(* IEC 61131-3 sources: std_i2980_v2.06_cp053/Source/IMM/ieccontrol/AutoPurgeGeneral, 3 files *)

(* ---- ABManualButton.pu ---- *)
(*

This postupdate algorithm reacts on changes of the autopurge button.
*)

IMPORT_OVER_LISTFILE
 cCompInjection
, tsMoveData
, FBManualButtonKeep
, tevPanelButtonRegister
, tsDeviceId
, tyPanelButton
, tevPanelButtonRegisterData
, tsPanelButton
, FBCheckReady

END_IMPORT

ALGORITHM_BLOCK ABManualButton #DUMMY_EDIT_BLOCK

SYSTEM_VAR
 sv_MoveAutoPurge : tsMoveData;
 di_ButtonAutoPurge : BOOL;
 sv_bInitStart : BOOL;
 sv_bButtonAutoPurge : BOOL;
 sv_bDeviceReady : BOOL;
 sv_bHMILedAutoPurge_ledAttr : BYTE (* Panel LED Attr *);
 sv_bHMILedAutoPurge : BOOL;
 sv_bLedAutoPurge_ledAttr : BYTE (* Panel LED Attr *);
 sv_bLedAutoPurge : BOOL;
 sv_bInitDone : BOOL;
 di_ButtonGeneral1 : BOOL;
 di_ButtonGeneral2 : BOOL;
 sv_iPanelMovementSelector : DINT;
 sv_DeviceId : tsDeviceId;
 sv_PanelButtons : tyPanelButton;
END_VAR

SYSTEM_OBJECT
 PU_Task_7 : TASK;
 PU_Task_13 : TASK;
 evPanelButtonRegister : tevPanelButtonRegister;
END_OBJECT

VAR
 fbManualButton : FBManualButtonKeep;
 mpbInjectionUnitReady : REFTO BOOL;
 evPanelButtonRegisterData : tevPanelButtonRegisterData;
 mpbButtonGeneralAutoPurge1 : REFTO BOOL;
 mpbButtonGeneralAutoPurge2 : REFTO BOOL;
 mbDIButtonAutoPurgeLinked : BOOL;
 mbDIButtonGeneral1Linked : BOOL;
 mbDIButtonGeneral2Linked : BOOL;
 mpiPanelMovementSelector : REFTO DINT;
END_VAR

VAR CONSTANT
 cButtonAutoPurge : DINT := 1;
END_VAR

ALGORITHM aButtonAutoPurge

VAR_INPUT
 bButton : BOOL;
END_VAR
#BEGIN_EDIT_BLOCK
(**************************************** WARNING ********************************************
 *** The KEBA Kemro K2 System including software is not intended for safety control tasks! ***
 ***                       For further information see Comment tab!                        ***
 *********************************************************************************************)

IF bButton AND sv_bDeviceReady AND mpbInjectionUnitReady <> EMPTY AND NOT mpbInjectionUnitReady^ THEN
    // purge should be started and movement of injection function unit active -> ignore manual button
    RETURN;
END_IF;

fbManualButton(bButton := bButton, MoveId := sv_MoveAutoPurge.MoveId, MoveDir := sv_MoveAutoPurge.MoveDir);

;#END_EDIT_BLOCK END_ALGORITHM

POSTUPDATE_ALGORITHM pButtonAutoPurge ON PU_Task_7 WITH di_ButtonAutoPurge,sv_bButtonAutoPurge,mpbButtonGeneralAutoPurge1^,mpbButtonGeneralAutoPurge2^

VAR
 bButton : BOOL;
END_VAR
#BEGIN_EDIT_BLOCK
(**************************************** WARNING ********************************************
 *** The KEBA Kemro K2 System including software is not intended for safety control tasks! ***
 ***                       For further information see Comment tab!                        ***
 *********************************************************************************************)

// soft panel button
bButton := sv_bButtonAutoPurge;

// hw panel button
IF mbDIButtonAutoPurgeLinked THEN
    bButton := bButton OR di_ButtonAutoPurge;
END_IF;

// external panel button
IF CHECK_REF(mpbButtonGeneralAutoPurge1^) THEN
    bButton := bButton OR mpbButtonGeneralAutoPurge1^;
END_IF;
IF CHECK_REF(mpbButtonGeneralAutoPurge2^) THEN
    bButton := bButton OR mpbButtonGeneralAutoPurge2^;
END_IF;

aButtonAutoPurge(bButton := bButton);

;#END_EDIT_BLOCK END_ALGORITHM

POSTUPDATE_ALGORITHM pRegisterButtons ON PU_Task_13 WITH sv_bInitStart

#BEGIN_EDIT_BLOCK
(**************************************** WARNING ********************************************
 *** The KEBA Kemro K2 System including software is not intended for safety control tasks! ***
 ***                       For further information see Comment tab!                        ***
 *********************************************************************************************)

mpbButtonGeneralAutoPurge1 := EMPTY;
mpbButtonGeneralAutoPurge2 := EMPTY;

mbDIButtonAutoPurgeLinked := IS_LINKED(di_ButtonAutoPurge);

mbDIButtonGeneral1Linked := IS_LINKED(di_ButtonGeneral1);
mbDIButtonGeneral2Linked := IS_LINKED(di_ButtonGeneral2);
IF (mbDIButtonGeneral1Linked AND mbDIButtonGeneral2Linked) THEN
    mpiPanelMovementSelector := @sv_iPanelMovementSelector;
END_IF;

evPanelButtonRegisterData.Button.nPanelButtonType := nPanelButtonMovement;
evPanelButtonRegisterData.Button.iCompId := sv_DeviceId.CompId;
evPanelButtonRegisterData.Button.iIndexId := sv_DeviceId.IndexId;
evPanelButtonRegisterData.Button.iButtonId := cButtonAutoPurge;
evPanelButtonRegisterData.Button.pbActionVar1 := @sv_bButtonAutoPurge;
evPanelButtonRegisterData.Button.pbActionVar2 := @sv_bButtonAutoPurge;
evPanelButtonRegisterData.Button.Optional.pbLedVar := @sv_bHMILedAutoPurge;
evPanelButtonRegisterData.Button.Optional.piLedVarAttr := @sv_bHMILedAutoPurge_ledAttr;

SET_EVENT(evPanelButtonRegister, evPanelButtonRegisterData);

;#END_EDIT_BLOCK END_ALGORITHM

POSTUPDATE_ALGORITHM pMoveSelectorChanged ON PU_Task_7 WITH mpiPanelMovementSelector^

VAR
 Button : tsPanelButton;
END_VAR
#BEGIN_EDIT_BLOCK
(**************************************** WARNING ********************************************
 *** The KEBA Kemro K2 System including software is not intended for safety control tasks! ***
 ***                       For further information see Comment tab!                        ***
 *********************************************************************************************)

mpbButtonGeneralAutoPurge1 := EMPTY;
mpbButtonGeneralAutoPurge2 := EMPTY;

IF (NOT sv_bDeviceReady) THEN
    // stop active movements
    aButtonAutoPurge(bButton := FALSE);
END_IF;

IF (sv_iPanelMovementSelector > 0) THEN
    Button := sv_PanelButtons[sv_iPanelMovementSelector];
    IF Button.iCompId = sv_DeviceId.CompId AND
        Button.iIndexId = sv_DeviceId.IndexId THEN

        IF Button.iButtonId = cButtonAutoPurge THEN
            mpbButtonGeneralAutoPurge1 := @di_ButtonGeneral1;
            mpbButtonGeneralAutoPurge2 := @di_ButtonGeneral2;
        END_IF;
    END_IF;
END_IF;

;#END_EDIT_BLOCK END_ALGORITHM

POSTUPDATE_ALGORITHM pLedControl ON PU_Task_7 WITH sv_bDeviceReady

VAR
 bInitDone : BOOL;
 mbLedAutoPurgeExists : BOOL := FALSE;
END_VAR
#BEGIN_EDIT_BLOCK
IF NOT bInitDone THEN
    sv_bHMILedAutoPurge_ledAttr := 16#3;
    IF IS_LINKED(sv_bLedAutoPurge) AND IS_LINKED(sv_bLedAutoPurge_ledAttr) THEN
        sv_bLedAutoPurge_ledAttr := sv_bHMILedAutoPurge_ledAttr;
        mbLedAutoPurgeExists := TRUE;
    ELSE
        mbLedAutoPurgeExists := FALSE;
    END_IF;

    bInitDone := TRUE;
END_IF;

IF NOT sv_bDeviceReady THEN
   //led should be on if purging is active
   sv_bHMILedAutoPurge := TRUE;
ELSE
   //switch off
   sv_bHMILedAutoPurge := FALSE;
END_IF;

IF mbLedAutoPurgeExists THEN
   sv_bLedAutoPurge := sv_bHMILedAutoPurge;
END_IF;

;#END_EDIT_BLOCK END_ALGORITHM

POSTUPDATE_ALGORITHM pInitDone ON PU_Task_7(10) WITH sv_bInitDone

VAR
 fbCheckInjectionReady : FBCheckReady;
 DeviceIdInjection : tsDeviceId;
END_VAR
#BEGIN_EDIT_BLOCK
(**************************************** WARNING ********************************************
 *** The KEBA Kemro K2 System including software is not intended for safety control tasks! ***
 ***                       For further information see Comment tab!                        ***
 *********************************************************************************************)

//get reference to ready flag of injection function unit
DeviceIdInjection.CompId := cCompInjection;
DeviceIdInjection.IndexId := sv_DeviceId.IndexId;

fbCheckInjectionReady(DeviceId := DeviceIdInjection);
mpbInjectionUnitReady := fbCheckInjectionReady.pbReady;

;#END_EDIT_BLOCK END_ALGORITHM

END_ALGORITHM_BLOCK

#END_OF_IEC_PART

@Puma @IecEditor 6 114 @Pou 25
@@@BEG_Comment@@@

This postupdate algorithm reacts on changes of the autopurge button.
@@@END_Comment@@@

@BEG_Contents

@BEG_Func
@RT(17)FuncTreeContainer
0
@END_Func

@BEG_Const
@RT(18)ConstTreeContainer
1
@Var @RT(14)cCompInjection @RT(0) @T @F @DT @RT(4)DINT @RT(0) @T @T @BASIC 0 @F
@F @F
@T
@BEG_Attrib
0 @RT(3)104 @RT(19)Component Injection
@END_Attrib
1 1 @F @F @F @F

@END_Const

@BEG_Export

@BEG_Kind
@ALGORITHM_BLOCK @RT(14)ABManualButton @STRUCTURED_TEXT
@RT(0) @RT(0) @RT(0)
@END_Kind

@BEG_Dcl
@RT(16)DclTreeContainer
28
@Var @RT(16)sv_MoveAutoPurge @RT(0) @T @T @DERIVED 0 @T @T @DT @RT(10)tsMoveData @RT(0) @T @T @UNKNOWN 0 @F
@F @F
@T
@BEG_Attrib
3 @RT(0) @RT(0) @RT(0)
@END_Attrib
1 8 @F @F @F @F

@Var @RT(18)di_ButtonAutoPurge @RT(0) @T @F @DT @RT(4)BOOL @RT(0) @T @T @BASIC 0 @F
@F @F
@T
@BEG_Attrib
3 @RT(0) @RT(0) @RT(0)
@END_Attrib
1 8 @F @F @F @F

@Var @RT(13)sv_bInitStart @RT(0) @T @F @DT @RT(4)BOOL @RT(0) @T @T @BASIC 0 @F
@F @F
@T
@BEG_Attrib
3 @RT(0) @RT(0) @RT(0)
@END_Attrib
1 8 @F @F @F @F

@Var @RT(19)sv_bButtonAutoPurge @RT(0) @T @F @DT @RT(4)BOOL @RT(0) @T @T @BASIC 0 @F
@F @F
@T
@BEG_Attrib
3 @RT(0) @RT(0) @RT(0)
@END_Attrib
1 8 @F @F @F @F

@Var @RT(15)sv_bDeviceReady @RT(0) @T @F @DT @RT(4)BOOL @RT(0) @T @T @BASIC 0 @F
@F @F
@T
@BEG_Attrib
3 @RT(0) @RT(0) @RT(0)
@END_Attrib
1 8 @F @F @F @F

@Var @RT(27)sv_bHMILedAutoPurge_ledAttr @RT(0) @T @F @DT @RT(4)BYTE @RT(0) @T @T @BASIC 0 @F
@F @F
@T
@BEG_Attrib
3 @RT(0) @RT(14)Panel LED Attr @RT(0)
@END_Attrib
1 8 @F @F @F @F

@Var @RT(19)sv_bHMILedAutoPurge @RT(0) @T @F @DT @RT(4)BOOL @RT(0) @T @T @BASIC 0 @F
@F @F
@T
@BEG_Attrib
3 @RT(0) @RT(0) @RT(0)
@END_Attrib
1 8 @F @F @F @F

@Var @RT(24)sv_bLedAutoPurge_ledAttr @RT(0) @T @F @DT @RT(4)BYTE @RT(0) @T @T @BASIC 0 @F
@F @F
@T
@BEG_Attrib
3 @RT(0) @RT(14)Panel LED Attr @RT(0)
@END_Attrib
1 8 @F @F @F @F

@Var @RT(16)sv_bLedAutoPurge @RT(0) @T @F @DT @RT(4)BOOL @RT(0) @T @T @BASIC 0 @F
@F @F
@T
@BEG_Attrib
3 @RT(0) @RT(0) @RT(0)
@END_Attrib
1 8 @F @F @F @F

@Var @RT(12)sv_bInitDone @RT(0) @T @F @DT @RT(4)BOOL @RT(0) @T @T @BASIC 0 @F
@F @F
@T
@BEG_Attrib
3 @RT(0) @RT(0) @RT(0)
@END_Attrib
1 8 @F @F @F @F

@Var @RT(9)PU_Task_7 @RT(0) @T @F @DT @RT(4)TASK @RT(0) @T @T @BASIC 0 @F
@F @F
@T
@BEG_Attrib
3 @RT(0) @RT(0) @RT(0)
@END_Attrib
1 7 @F @F @F @F

@Var @RT(10)PU_Task_13 @RT(0) @T @F @DT @RT(4)TASK @RT(0) @T @T @BASIC 0 @F
@F @F
@T
@BEG_Attrib
3 @RT(0) @RT(0) @RT(0)
@END_Attrib
1 7 @F @F @F @F

@Var @RT(14)fbManualButton @RT(0) @T @T @DERIVED 0 @T @T @DT @RT(18)FBManualButtonKeep @RT(0) @T @T @UNKNOWN 0 @F
@F @F
@T
@BEG_Attrib
3 @RT(0) @RT(0) @RT(0)
@END_Attrib
1 0 @F @F @F @F

@Var @RT(21)mpbInjectionUnitReady @RT(0) @T @T @REFTO 0 @T @DT @RT(4)BOOL @RT(0) @T @T @BASIC 0 @F
@F @F
@T
@BEG_Attrib
3 @RT(0) @RT(0) @RT(0)
@END_Attrib
1 0 @F @F @F @F

@Var @RT(21)evPanelButtonRegister @RT(0) @T @T @DERIVED 0 @T @T @DT @RT(22)tevPanelButtonRegister @RT(0) @T @T @UNKNOWN 0 @F
@F @F
@T
@BEG_Attrib
3 @RT(0) @RT(0) @RT(0)
@END_Attrib
1 7 @F @F @F @F

@Var @RT(17)di_ButtonGeneral1 @RT(0) @T @F @DT @RT(4)BOOL @RT(0) @T @T @BASIC 0 @F
@F @F
@T
@BEG_Attrib
3 @RT(0) @RT(0) @RT(0)
@END_Attrib
1 8 @F @F @F @F

@Var @RT(17)di_ButtonGeneral2 @RT(0) @T @F @DT @RT(4)BOOL @RT(0) @T @T @BASIC 0 @F
@F @F
@T
@BEG_Attrib
3 @RT(0) @RT(0) @RT(0)
@END_Attrib
1 8 @F @F @F @F

@Var @RT(25)sv_iPanelMovementSelector @RT(0) @T @F @DT @RT(4)DINT @RT(0) @T @T @BASIC 0 @F
@F @F
@T
@BEG_Attrib
3 @RT(0) @RT(0) @RT(0)
@END_Attrib
1 8 @F @F @F @F

@Var @RT(11)sv_DeviceId @RT(0) @T @T @DERIVED 0 @T @T @DT @RT(10)tsDeviceId @RT(0) @T @T @UNKNOWN 0 @F
@F @F
@T
@BEG_Attrib
3 @RT(0) @RT(0) @RT(0)
@END_Attrib
1 8 @F @F @F @F

@Var @RT(15)sv_PanelButtons @RT(0) @T @T @DERIVED 0 @T @T @DT @RT(13)tyPanelButton @RT(0) @T @T @UNKNOWN 0 @F
@F @F
@T
@BEG_Attrib
3 @RT(0) @RT(0) @RT(0)
@END_Attrib
1 8 @F @F @F @F

@Var @RT(25)evPanelButtonRegisterData @RT(0) @T @T @DERIVED 0 @T @T @DT @RT(26)tevPanelButtonRegisterData @RT(0) @T @T @UNKNOWN 0 @F
@F @F
@T
@BEG_Attrib
3 @RT(0) @RT(0) @RT(0)
@END_Attrib
1 0 @F @F @F @F

@Var @RT(26)mpbButtonGeneralAutoPurge1 @RT(0) @T @T @REFTO 0 @T @DT @RT(4)BOOL @RT(0) @T @T @BASIC 0 @F
@F @F
@T
@BEG_Attrib
3 @RT(0) @RT(0) @RT(0)
@END_Attrib
1 0 @F @F @F @F

@Var @RT(26)mpbButtonGeneralAutoPurge2 @RT(0) @T @T @REFTO 0 @T @DT @RT(4)BOOL @RT(0) @T @T @BASIC 0 @F
@F @F
@T
@BEG_Attrib
3 @RT(0) @RT(0) @RT(0)
@END_Attrib
1 0 @F @F @F @F

@Var @RT(25)mbDIButtonAutoPurgeLinked @RT(0) @T @F @DT @RT(4)BOOL @RT(0) @T @T @BASIC 0 @F
@F @F
@T
@BEG_Attrib
3 @RT(0) @RT(0) @RT(0)
@END_Attrib
1 0 @F @F @F @F

@Var @RT(24)mbDIButtonGeneral1Linked @RT(0) @T @F @DT @RT(4)BOOL @RT(0) @T @T @BASIC 0 @F
@F @F
@T
@BEG_Attrib
3 @RT(0) @RT(0) @RT(0)
@END_Attrib
1 0 @F @F @F @F

@Var @RT(24)mbDIButtonGeneral2Linked @RT(0) @T @F @DT @RT(4)BOOL @RT(0) @T @T @BASIC 0 @F
@F @F
@T
@BEG_Attrib
3 @RT(0) @RT(0) @RT(0)
@END_Attrib
1 0 @F @F @F @F

@Var @RT(16)cButtonAutoPurge @RT(0) @T @F @DT @RT(4)DINT @RT(0) @T @T @BASIC 0 @F
@F @F
@T
@BEG_Attrib
3 @RT(1)1 @RT(0) @RT(0)
@END_Attrib
1 15 @F @F @F @F

@Var @RT(24)mpiPanelMovementSelector @RT(0) @T @T @REFTO 0 @T @DT @RT(4)DINT @RT(0) @T @T @BASIC 0 @F
@F @F
@T
@BEG_Attrib
3 @RT(0) @RT(0) @RT(0)
@END_Attrib
1 0 @F @F @F @F

@END_Dcl

@END_Export

@BEG_Body

6

@BEG_Export

@BEG_Algo
@ALGORITHM @RT(16)aButtonAutoPurge @STRUCTURED_TEXT
@RT(0) @RT(0) @RT(0) @F @F
@END_Algo

@BEG_Dcl
@RT(16)DclTreeContainer
1
@Var @RT(7)bButton @RT(0) @T @F @DT @RT(4)BOOL @RT(0) @T @T @BASIC 0 @F
@F @F
@T
@BEG_Attrib
3 @RT(0) @RT(0) @RT(0)
@END_Attrib
1 1 @F @F @F @F

@END_Dcl

@END_Export

@BEG_Export

@BEG_Algo
@POSTUPDATE_ALGORITHM @RT(16)pButtonAutoPurge @STRUCTURED_TEXT
@RT(0) @RT(94)di_ButtonAutoPurge,sv_bButtonAutoPurge,mpbButtonGeneralAutoPurge1^,mpbButtonGeneralAutoPurge2^ @RT(9)PU_Task_7 @F @F
@END_Algo

@BEG_Dcl
@RT(16)DclTreeContainer
1
@Var @RT(7)bButton @RT(0) @T @F @DT @RT(4)BOOL @RT(0) @T @T @BASIC 0 @F
@F @F
@T
@BEG_Attrib
3 @RT(0) @RT(0) @RT(0)
@END_Attrib
1 0 @F @F @F @F

@END_Dcl

@END_Export

@BEG_Export

@BEG_Algo
@POSTUPDATE_ALGORITHM @RT(16)pRegisterButtons @STRUCTURED_TEXT
@RT(0) @RT(13)sv_bInitStart @RT(10)PU_Task_13 @F @F
@END_Algo

@BEG_Dcl
@RT(16)DclTreeContainer
0
@END_Dcl

@END_Export

@BEG_Export

@BEG_Algo
@POSTUPDATE_ALGORITHM @RT(20)pMoveSelectorChanged @STRUCTURED_TEXT
@RT(0) @RT(25)mpiPanelMovementSelector^ @RT(9)PU_Task_7 @F @F
@END_Algo

@BEG_Dcl
@RT(16)DclTreeContainer
1
@Var @RT(6)Button @RT(0) @T @T @DERIVED 0 @T @T @DT @RT(13)tsPanelButton @RT(0) @T @T @UNKNOWN 0 @F
@F @F
@T
@BEG_Attrib
3 @RT(0) @RT(0) @RT(0)
@END_Attrib
1 0 @F @F @F @F

@END_Dcl

@END_Export

@BEG_Export

@BEG_Algo
@POSTUPDATE_ALGORITHM @RT(11)pLedControl @STRUCTURED_TEXT
@RT(0) @RT(15)sv_bDeviceReady @RT(9)PU_Task_7 @F @F
@END_Algo

@BEG_Dcl
@RT(16)DclTreeContainer
2
@Var @RT(9)bInitDone @RT(0) @T @F @DT @RT(4)BOOL @RT(0) @T @T @BASIC 0 @F
@F @F
@T
@BEG_Attrib
3 @RT(0) @RT(0) @RT(0)
@END_Attrib
1 0 @F @F @F @F

@Var @RT(20)mbLedAutoPurgeExists @RT(0) @T @F @DT @RT(4)BOOL @RT(0) @T @T @BASIC 0 @F
@F @F
@T
@BEG_Attrib
3 @RT(5)FALSE @RT(0) @RT(0)
@END_Attrib
1 0 @F @F @F @F

@END_Dcl

@END_Export

@BEG_Export

@BEG_Algo
@POSTUPDATE_ALGORITHM @RT(9)pInitDone @STRUCTURED_TEXT
@RT(0) @RT(12)sv_bInitDone @RT(13)PU_Task_7(10) @F @F
@END_Algo

@BEG_Dcl
@RT(16)DclTreeContainer
2
@Var @RT(21)fbCheckInjectionReady @RT(0) @T @T @DERIVED 0 @T @T @DT @RT(12)FBCheckReady @RT(0) @T @T @UNKNOWN 0 @F
@F @F
@T
@BEG_Attrib
3 @RT(0) @RT(0) @RT(0)
@END_Attrib
1 0 @F @F @F @F

@Var @RT(17)DeviceIdInjection @RT(0) @T @T @DERIVED 0 @T @T @DT @RT(10)tsDeviceId @RT(0) @T @T @UNKNOWN 0 @F
@F @F
@T
@BEG_Attrib
3 @RT(0) @RT(0) @RT(0)
@END_Attrib
1 0 @F @F @F @F

@END_Dcl

@END_Export

@BEG_Body
@TL(13)
(**************************************** WARNING ********************************************
 *** The KEBA Kemro K2 System including software is not intended for safety control tasks! ***
 ***                       For further information see Comment tab!                        ***
 *********************************************************************************************)

IF bButton AND sv_bDeviceReady AND mpbInjectionUnitReady <> EMPTY AND NOT mpbInjectionUnitReady^ THEN
    // purge should be started and movement of injection function unit active -> ignore manual button
    RETURN;
END_IF;

fbManualButton(bButton := bButton, MoveId := sv_MoveAutoPurge.MoveId, MoveDir := sv_MoveAutoPurge.MoveDir);

@END_Body

@@@BEG_Comment@@@
@TL(0)

@@@END_Comment@@@

@BEG_Body
@TL(24)
(**************************************** WARNING ********************************************
 *** The KEBA Kemro K2 System including software is not intended for safety control tasks! ***
 ***                       For further information see Comment tab!                        ***
 *********************************************************************************************)

// soft panel button
bButton := sv_bButtonAutoPurge;

// hw panel button
IF mbDIButtonAutoPurgeLinked THEN
    bButton := bButton OR di_ButtonAutoPurge;
END_IF;

// external panel button
IF CHECK_REF(mpbButtonGeneralAutoPurge1^) THEN
    bButton := bButton OR mpbButtonGeneralAutoPurge1^;
END_IF;
IF CHECK_REF(mpbButtonGeneralAutoPurge2^) THEN
    bButton := bButton OR mpbButtonGeneralAutoPurge2^;
END_IF;

aButtonAutoPurge(bButton := bButton);

@END_Body

@@@BEG_Comment@@@
@TL(0)

@@@END_Comment@@@

@BEG_Body
@TL(27)
(**************************************** WARNING ********************************************
 *** The KEBA Kemro K2 System including software is not intended for safety control tasks! ***
 ***                       For further information see Comment tab!                        ***
 *********************************************************************************************)

mpbButtonGeneralAutoPurge1 := EMPTY;
mpbButtonGeneralAutoPurge2 := EMPTY;

mbDIButtonAutoPurgeLinked := IS_LINKED(di_ButtonAutoPurge);

mbDIButtonGeneral1Linked := IS_LINKED(di_ButtonGeneral1);
mbDIButtonGeneral2Linked := IS_LINKED(di_ButtonGeneral2);
IF (mbDIButtonGeneral1Linked AND mbDIButtonGeneral2Linked) THEN
    mpiPanelMovementSelector := @sv_iPanelMovementSelector;
END_IF;

evPanelButtonRegisterData.Button.nPanelButtonType := nPanelButtonMovement;
evPanelButtonRegisterData.Button.iCompId := sv_DeviceId.CompId;
evPanelButtonRegisterData.Button.iIndexId := sv_DeviceId.IndexId;
evPanelButtonRegisterData.Button.iButtonId := cButtonAutoPurge;
evPanelButtonRegisterData.Button.pbActionVar1 := @sv_bButtonAutoPurge;
evPanelButtonRegisterData.Button.pbActionVar2 := @sv_bButtonAutoPurge;
evPanelButtonRegisterData.Button.Optional.pbLedVar := @sv_bHMILedAutoPurge;
evPanelButtonRegisterData.Button.Optional.piLedVarAttr := @sv_bHMILedAutoPurge_ledAttr;

SET_EVENT(evPanelButtonRegister, evPanelButtonRegisterData);

@END_Body

@@@BEG_Comment@@@
@TL(0)

@@@END_Comment@@@

@BEG_Body
@TL(26)
(**************************************** WARNING ********************************************
 *** The KEBA Kemro K2 System including software is not intended for safety control tasks! ***
 ***                       For further information see Comment tab!                        ***
 *********************************************************************************************)

mpbButtonGeneralAutoPurge1 := EMPTY;
mpbButtonGeneralAutoPurge2 := EMPTY;

IF (NOT sv_bDeviceReady) THEN
    // stop active movements
    aButtonAutoPurge(bButton := FALSE);
END_IF;

IF (sv_iPanelMovementSelector > 0) THEN
    Button := sv_PanelButtons[sv_iPanelMovementSelector];
    IF Button.iCompId = sv_DeviceId.CompId AND
        Button.iIndexId = sv_DeviceId.IndexId THEN

        IF Button.iButtonId = cButtonAutoPurge THEN
            mpbButtonGeneralAutoPurge1 := @di_ButtonGeneral1;
            mpbButtonGeneralAutoPurge2 := @di_ButtonGeneral2;
        END_IF;
    END_IF;
END_IF;

@END_Body

@@@BEG_Comment@@@
@TL(0)

@@@END_Comment@@@

@BEG_Body
@TL(26)
IF NOT bInitDone THEN
    sv_bHMILedAutoPurge_ledAttr := 16#3;
    IF IS_LINKED(sv_bLedAutoPurge) AND IS_LINKED(sv_bLedAutoPurge_ledAttr) THEN
        sv_bLedAutoPurge_ledAttr := sv_bHMILedAutoPurge_ledAttr;
        mbLedAutoPurgeExists := TRUE;
    ELSE
        mbLedAutoPurgeExists := FALSE;
    END_IF;

    bInitDone := TRUE;
END_IF;

IF NOT sv_bDeviceReady THEN
   //led should be on if purging is active
   sv_bHMILedAutoPurge := TRUE;
ELSE
   //switch off
   sv_bHMILedAutoPurge := FALSE;
END_IF;

IF mbLedAutoPurgeExists THEN
   sv_bLedAutoPurge := sv_bHMILedAutoPurge;
END_IF;

@END_Body

@@@BEG_Comment@@@
@TL(0)

@@@END_Comment@@@

@BEG_Body
@TL(13)
(**************************************** WARNING ********************************************
 *** The KEBA Kemro K2 System including software is not intended for safety control tasks! ***
 ***                       For further information see Comment tab!                        ***
 *********************************************************************************************)

//get reference to ready flag of injection function unit
DeviceIdInjection.CompId := cCompInjection;
DeviceIdInjection.IndexId := sv_DeviceId.IndexId;

fbCheckInjectionReady(DeviceId := DeviceIdInjection);
mpbInjectionUnitReady := fbCheckInjectionReady.pbReady;

@END_Body

@@@BEG_Comment@@@
@TL(0)

@@@END_Comment@@@
@END_Body

@END_Contents

(* ---- ABMoveAutoPurge.pu ---- *)
(*

@FunctionID: S_KPIEC_PRINJ_03

*)

IMPORT_OVER_LISTFILE
 SET_EVENT
, cLockGroupHeatingNozzle
, cLockGroupSafetyGateNozzle
, cLockGroupSafetyGateMold
, cLockGroupMotor
, cCompInjection
, cMoveFwd
, cMoveInjectPurge
, cMoveBwd
, cMoveDecompPurge
, cMovePlastPurge
, cCompShutOffNozzle
, cMoveClose
, cMoveOpen
, tsMoveData
, tsPurgeSettings
, tsActPurgeTimes
, tyNumberOfDevices
, tsDeviceId
, tevStartRequest
, ABMovementRegister
, tevStartRequestData
, FBCheckReady
, FBStop
, FBCheckPosReached
, FBDebugTrace2

END_IMPORT

ALGORITHM_BLOCK ABMoveAutoPurge #DUMMY_EDIT_BLOCK

SYSTEM_VAR
 sv_MoveAutoPurge : tsMoveData;
 sv_PurgeSettings : tsPurgeSettings;
 sv_rScrewPosition : REAL (* actual screw position *);
 sv_ActPurgeTimes : tsActPurgeTimes;
 sv_NumberOfDevices : tyNumberOfDevices;
 sv_DeviceId : tsDeviceId;
END_VAR

SYSTEM_OBJECT
 evStartRequest : tevStartRequest;
END_OBJECT

ALGORITHM aRegister

VAR
 abMovementRegister : ABMovementRegister;
END_VAR
#BEGIN_EDIT_BLOCK
(**************************************** WARNING ********************************************
 *** The KEBA Kemro K2 System including software is not intended for safety control tasks! ***
 ***                       For further information see Comment tab!                        ***
 *********************************************************************************************)

// movement registration
sv_MoveAutoPurge.LockGroups[1] := cLockGroupHeatingNozzle;
sv_MoveAutoPurge.LockGroups[2] := cLockGroupSafetyGateNozzle;
sv_MoveAutoPurge.LockGroups[3] := cLockGroupSafetyGateMold;
sv_MoveAutoPurge.LockGroups[4] := cLockGroupMotor;

abMovementRegister.aRegister(@sv_MoveAutoPurge);

;#END_EDIT_BLOCK END_ALGORITHM

ALGORITHM aRun

VAR_OUTPUT
 bReady : BOOL;
END_VAR

VAR_INPUT
 bStop : BOOL;
END_VAR

VAR
 evStartRequestData : tevStartRequestData;
 DeviceId : tsDeviceId;
 fbCheckReady : FBCheckReady;
 iCount : DINT;
 fbStop : FBStop;
 bShutOffNozzleAvailable : BOOL;
 bInitDone : BOOL;
 pbShutOffNozzleOpen : REFTO BOOL;
 pbShutOffNozzleClosed : REFTO BOOL;
 DeviceIdShutOffNozzle : tsDeviceId;
 fbCheckPosReached : FBCheckPosReached;
 fbDebugTrace2 : FBDebugTrace2;
 dTmpPurgePlastTime : TIME;
 rTmpPurgeDecompPos : REAL;
END_VAR

(* IecGraph-Code *)

(* init step *)
INITIAL_STEP S_Start:
AInitShutOffNozzle (P);
AStart (P);
END_STEP

ACTION AStart: #BEGIN_EDIT_BLOCK
bReady := FALSE;
fbDebugTrace2(nDeviceState, 'AutoPurge started');
iCount := 0;

;#END_EDIT_BLOCK END_ACTION (*AStart*)

(* steps *)
STEP Step17:
END_STEP

STEP S_OpenShutOffNozzle:
AStartOpen (P);
ACheckShutOffNozzle (N);
END_STEP

ACTION ACheckShutOffNozzle: #BEGIN_EDIT_BLOCK
fbCheckReady(DeviceId := DeviceId);

;#END_EDIT_BLOCK END_ACTION (*ACheckShutOffNozzle*)
STEP S_Inject:
AStartInject (P);
ACheckInjectReady (N);
END_STEP

ACTION AStartInject: #BEGIN_EDIT_BLOCK
// send start request
DeviceId.CompId := cCompInjection;
DeviceId.IndexId := sv_DeviceId.IndexId;

evStartRequestData.DeviceId := DeviceId;
evStartRequestData.MoveDir := cMoveFwd;
evStartRequestData.MoveId := cMoveInjectPurge;
SET_EVENT(evStartRequest, evStartRequestData);

;#END_EDIT_BLOCK END_ACTION (*AStartInject*)
ACTION ACheckInjectReady: #BEGIN_EDIT_BLOCK
fbCheckReady(DeviceId := DeviceId);

;#END_EDIT_BLOCK END_ACTION (*ACheckInjectReady*)
STEP S_Decomp:
AStartDecomp (P);
ACheckDecompReady (N);
END_STEP

ACTION AStartDecomp: #BEGIN_EDIT_BLOCK
//copy decomp position to avoid wrongly detecting a error
//when the value changes while the movement is active
rTmpPurgeDecompPos := sv_PurgeSettings.DecompParams.rEndPos;

// send start request
DeviceId.CompId := cCompInjection;
DeviceId.IndexId := sv_DeviceId.IndexId;

evStartRequestData.DeviceId := DeviceId;
evStartRequestData.MoveDir := cMoveBwd;
evStartRequestData.MoveId := cMoveDecompPurge;
SET_EVENT(evStartRequest, evStartRequestData);

;#END_EDIT_BLOCK END_ACTION (*AStartDecomp*)
ACTION ACheckDecompReady: #BEGIN_EDIT_BLOCK
fbCheckReady(DeviceId := DeviceId);

;#END_EDIT_BLOCK END_ACTION (*ACheckDecompReady*)
STEP S_Plast:
AStartPlast (P);
ACheckPlastReady (N);
END_STEP

ACTION AStartPlast: #BEGIN_EDIT_BLOCK
//copy purge set time to avoid wrongly detecting a error
//when the value changes while the movement is active
dTmpPurgePlastTime := sv_PurgeSettings.PlastParams.dSetPlastTime;

// send start request
DeviceId.CompId := cCompInjection;
DeviceId.IndexId := sv_DeviceId.IndexId;

evStartRequestData.DeviceId := DeviceId;
evStartRequestData.MoveDir := cMoveBwd;
evStartRequestData.MoveId := cMovePlastPurge;
SET_EVENT(evStartRequest, evStartRequestData);

;#END_EDIT_BLOCK END_ACTION (*AStartPlast*)
ACTION ACheckPlastReady: #BEGIN_EDIT_BLOCK
fbCheckReady(DeviceId := DeviceId);

;#END_EDIT_BLOCK END_ACTION (*ACheckPlastReady*)
STEP S_CheckCounter:
ACounter (P);
END_STEP

ACTION ACounter: #BEGIN_EDIT_BLOCK
iCount := iCount + 1;

;#END_EDIT_BLOCK END_ACTION (*ACounter*)
STEP S_CheckStop:
END_STEP

STEP S_Stop:
AStopActiveMovement (P);
AStoppedMoveReady (N);
END_STEP

ACTION AStopActiveMovement: #BEGIN_EDIT_BLOCK
//stop actual active movement
fbStop(DeviceId := DeviceId);

;#END_EDIT_BLOCK END_ACTION (*AStopActiveMovement*)
ACTION AStoppedMoveReady: #BEGIN_EDIT_BLOCK
fbCheckReady(DeviceId := DeviceId);

;#END_EDIT_BLOCK END_ACTION (*AStoppedMoveReady*)
STEP Step27:
END_STEP

STEP S_CloseShutOffNozzle:
AStartClose (P);
ACheckShutOff (N);
END_STEP

ACTION ACheckShutOff: #BEGIN_EDIT_BLOCK
fbCheckReady(DeviceId := DeviceId);

;#END_EDIT_BLOCK END_ACTION (*ACheckShutOff*)
STEP S_Ready:
AReady (P);
END_STEP

ACTION AReady: #BEGIN_EDIT_BLOCK
bReady := TRUE;
fbDebugTrace2(nDeviceState, 'AutoPurge ready');

;#END_EDIT_BLOCK END_ACTION (*AReady*)

(* transitions *)
GO_ON_TRANSITION TStart (* Trans21 *) FROM S_Start TO Step17 :=  #BEGIN_EDIT_BLOCK
TRUE
;#END_EDIT_BLOCK
END_TRANSITION

GO_ON_TRANSITION TShutOffNozzle (* TShutOffNozzle *) FROM Step17 TO S_OpenShutOffNozzle :=  #BEGIN_EDIT_BLOCK
bShutOffNozzleAvailable
;#END_EDIT_BLOCK
END_TRANSITION

TRANSITION TShutOffNozzleOpen (* TShutOffNozzleOpen *) FROM S_OpenShutOffNozzle TO S_Inject :=  #BEGIN_EDIT_BLOCK
fbCheckReady.bReady AND pbShutOffNozzleOpen^
;#END_EDIT_BLOCK
END_TRANSITION

TRANSITION TStop4 (* TStop4 *) FROM S_OpenShutOffNozzle TO S_Stop :=  #BEGIN_EDIT_BLOCK
bStop
;#END_EDIT_BLOCK
END_TRANSITION

GO_ON_TRANSITION TNoShutOffNozzle (* TNoShutOffNozzle *) FROM Step17 TO S_Inject :=  #BEGIN_EDIT_BLOCK
NOT bShutOffNozzleAvailable
;#END_EDIT_BLOCK
END_TRANSITION

TRANSITION TInjectReady (* TInjectReady *) FROM S_Inject TO S_Decomp :=  #BEGIN_EDIT_BLOCK
fbCheckReady.bReady AND
sv_rScrewPosition <= sv_PurgeSettings.InjectParams.rEndPos
;#END_EDIT_BLOCK
END_TRANSITION

TRANSITION TStop1 (* TStop1 *) FROM S_Inject TO S_Stop :=  #BEGIN_EDIT_BLOCK
bStop
;#END_EDIT_BLOCK
END_TRANSITION

TRANSITION TDecompReady (* TDecompReady *) FROM S_Decomp TO S_Plast :=  #BEGIN_EDIT_BLOCK
fbCheckReady.bReady AND
sv_rScrewPosition >= rTmpPurgeDecompPos
;#END_EDIT_BLOCK
END_TRANSITION

TRANSITION TStop2 (* TStop2 *) FROM S_Decomp TO S_Stop :=  #BEGIN_EDIT_BLOCK
bStop
;#END_EDIT_BLOCK
END_TRANSITION

TRANSITION TPlastReady (* TPlastReady *) FROM S_Plast TO S_CheckCounter :=  #BEGIN_EDIT_BLOCK
fbCheckReady.bReady AND
sv_ActPurgeTimes.dActPlastTime >= dTmpPurgePlastTime
;#END_EDIT_BLOCK
END_TRANSITION

TRANSITION TStop3 (* TStop3 *) FROM S_Plast TO S_Stop :=  #BEGIN_EDIT_BLOCK
bStop
;#END_EDIT_BLOCK
END_TRANSITION

GO_ON_TRANSITION TRepeat (* TRepeat *) FROM S_CheckCounter TO S_Inject :=  #BEGIN_EDIT_BLOCK
iCount < sv_PurgeSettings.iCount
;#END_EDIT_BLOCK
END_TRANSITION

GO_ON_TRANSITION TReady (* TReady *) FROM S_CheckCounter TO S_CheckStop :=  #BEGIN_EDIT_BLOCK
iCount = sv_PurgeSettings.iCount
;#END_EDIT_BLOCK
END_TRANSITION

GO_ON_TRANSITION TStop (* TStop *) FROM S_CheckStop TO S_Stop :=  #BEGIN_EDIT_BLOCK
bStop
;#END_EDIT_BLOCK
END_TRANSITION

TRANSITION TStoppedDeviceReady (* TStoppedDeviceReady *) FROM S_Stop TO Step27 :=  #BEGIN_EDIT_BLOCK
fbCheckReady.bReady
;#END_EDIT_BLOCK
END_TRANSITION

GO_ON_TRANSITION TNoStop (* TNoStop *) FROM S_CheckStop TO Step27 :=  #BEGIN_EDIT_BLOCK
NOT bStop
;#END_EDIT_BLOCK
END_TRANSITION

GO_ON_TRANSITION Trans36 (* Trans36 *) FROM Step27 TO S_CloseShutOffNozzle :=  #BEGIN_EDIT_BLOCK
bShutOffNozzleAvailable
;#END_EDIT_BLOCK
END_TRANSITION

TRANSITION TShutOffNozzleReady (* TShutOffNozzleClosed *) FROM S_CloseShutOffNozzle TO S_Ready :=  #BEGIN_EDIT_BLOCK
fbCheckReady.bReady
;#END_EDIT_BLOCK
END_TRANSITION

GO_ON_TRANSITION Trans37 (* Trans37 *) FROM Step27 TO S_Ready :=  #BEGIN_EDIT_BLOCK
NOT bShutOffNozzleAvailable
;#END_EDIT_BLOCK
END_TRANSITION

TRANSITION Trans12 (* Trans12 *) FROM S_Ready TO S_Start :=  #BEGIN_EDIT_BLOCK
TRUE
;#END_EDIT_BLOCK
END_TRANSITION

(* end IecGraph-Code *)
(* sfc-code *)

(* stand alone actions *)
ACTION AInitShutOffNozzle: #BEGIN_EDIT_BLOCK
//check if shut off nozzle is available
IF NOT bInitDone THEN
   bShutOffNozzleAvailable := sv_NumberOfDevices[cCompShutOffNozzle] = sv_DeviceId.IndexId;
END_IF;

IF bShutOffNozzleAvailable AND NOT bInitDone THEN
   //get pos reached flags of shut off nozzle
   DeviceIdShutOffNozzle.CompId := cCompShutOffNozzle;
   DeviceIdShutOffNozzle.IndexId := sv_DeviceId.IndexId;

   fbCheckPosReached.DeviceId := DeviceIdShutOffNozzle;
   fbCheckPosReached.MoveDir := cMoveClose;
   fbCheckPosReached.MoveId := cMoveClose;
   fbCheckPosReached();
   pbShutOffNozzleClosed := fbCheckPosReached.pbPosReached;

   fbCheckPosReached.MoveDir := cMoveOpen;
   fbCheckPosReached.MoveId := cMoveOpen;
   fbCheckPosReached();
   pbShutOffNozzleOpen := fbCheckPosReached.pbPosReached;
END_IF;

bInitDone := TRUE;

;#END_EDIT_BLOCK END_ACTION (*AInitShutOffNozzle*)
ACTION AStartOpen: #BEGIN_EDIT_BLOCK
(**************************************** WARNING ********************************************
 *** The KEBA Kemro K2 System including software is not intended for safety control tasks! ***
 ***                       For further information see Comment tab!                        ***
 *********************************************************************************************)

// send start request
DeviceId := DeviceIdShutOffNozzle;

evStartRequestData.DeviceId := DeviceId;
evStartRequestData.MoveDir := cMoveOpen;
evStartRequestData.MoveId := cMoveOpen;
SET_EVENT(evStartRequest, evStartRequestData);

;#END_EDIT_BLOCK END_ACTION (*AStartOpen*)
ACTION AStartClose: #BEGIN_EDIT_BLOCK
(**************************************** WARNING ********************************************
 *** The KEBA Kemro K2 System including software is not intended for safety control tasks! ***
 ***                       For further information see Comment tab!                        ***
 *********************************************************************************************)

// send start request
DeviceId := DeviceIdShutOffNozzle;
evStartRequestData.DeviceId := DeviceId;
evStartRequestData.MoveDir := cMoveClose;
evStartRequestData.MoveId := cMoveClose;
SET_EVENT(evStartRequest, evStartRequestData);

;#END_EDIT_BLOCK END_ACTION (*AStartClose*)
(* end sfc-code *)

END_ALGORITHM

END_ALGORITHM_BLOCK

#END_OF_IEC_PART

@Puma @IecEditor 6 103 @Pou 25
@@@BEG_Comment@@@

@FunctionID: S_KPIEC_PRINJ_03

@@@END_Comment@@@

@BEG_Contents

@BEG_Func
@RT(17)FuncTreeContainer
1
@Var @RT(9)SET_EVENT @RT(0) @T @T @DERIVED 0 @F @RT(23)KEBA_STANDARD_PROCEDURE @F
@T
@BEG_Attrib
0 @RT(0) @RT(0)
@END_Attrib
1 1 @F @F @F @F

@END_Func

@BEG_Const
@RT(18)ConstTreeContainer
13
@Var @RT(23)cLockGroupHeatingNozzle @RT(0) @T @F @DT @RT(4)DINT @RT(0) @T @T @BASIC 0 @F
@F @F
@T
@BEG_Attrib
0 @RT(2)63 @RT(35)Members: Injection, Plast, Suckback
@END_Attrib
1 1 @F @F @F @F

@Var @RT(26)cLockGroupSafetyGateNozzle @RT(0) @T @F @DT @RT(4)DINT @RT(0) @T @T @BASIC 0 @F
@F @F
@T
@BEG_Attrib
0 @RT(2)62 @RT(59)Members: Nozzle Forward, Injection, Plast, Intrusion, Purge
@END_Attrib
1 1 @F @F @F @F

@Var @RT(24)cLockGroupSafetyGateMold @RT(0) @T @F @DT @RT(4)DINT @RT(0) @T @T @BASIC 0 @F
@F @F
@T
@BEG_Attrib
0 @RT(2)61 @RT(73)Members: Mold Close, Mold Hight Forward, Auto Mold Hight, Core In, Inject
@END_Attrib
1 1 @F @F @F @F

@Var @RT(15)cLockGroupMotor @RT(0) @T @F @DT @RT(4)DINT @RT(0) @T @T @BASIC 0 @F
@F @F
@T
@BEG_Attrib
0 @RT(2)69 @RT(56)Members: Mold, Ejector, Cores, Injection, Plast, Purge,
@END_Attrib
1 1 @F @F @F @F

@Var @RT(14)cCompInjection @RT(0) @T @F @DT @RT(4)DINT @RT(0) @T @T @BASIC 0 @F
@F @F
@T
@BEG_Attrib
0 @RT(3)104 @RT(19)Component Injection
@END_Attrib
1 1 @F @F @F @F

@Var @RT(8)cMoveFwd @RT(0) @T @F @DT @RT(4)DINT @RT(0) @T @T @BASIC 0 @F
@F @F
@T
@BEG_Attrib
0 @RT(2)12 @RT(16)movement forward
@END_Attrib
1 1 @F @F @F @F

@Var @RT(16)cMoveInjectPurge @RT(0) @T @F @DT @RT(4)DINT @RT(0) @T @T @BASIC 0 @F
@F @F
@T
@BEG_Attrib
0 @RT(2)35 @RT(27)inject movement for purging
@END_Attrib
1 1 @F @F @F @F

@Var @RT(8)cMoveBwd @RT(0) @T @F @DT @RT(4)DINT @RT(0) @T @T @BASIC 0 @F
@F @F
@T
@BEG_Attrib
0 @RT(2)11 @RT(17)movement backward
@END_Attrib
1 1 @F @F @F @F

@Var @RT(16)cMoveDecompPurge @RT(0) @T @F @DT @RT(4)DINT @RT(0) @T @T @BASIC 0 @F
@F @F
@T
@BEG_Attrib
0 @RT(2)36 @RT(27)decomp movement for purging
@END_Attrib
1 1 @F @F @F @F

@Var @RT(15)cMovePlastPurge @RT(0) @T @F @DT @RT(4)DINT @RT(0) @T @T @BASIC 0 @F
@F @F
@T
@BEG_Attrib
0 @RT(2)34 @RT(26)plast movement for purging
@END_Attrib
1 1 @F @F @F @F

@Var @RT(18)cCompShutOffNozzle @RT(0) @T @F @DT @RT(4)DINT @RT(0) @T @T @BASIC 0 @F
@F @F
@T
@BEG_Attrib
0 @RT(3)138 @RT(28)Component Shutter for Nozzle
@END_Attrib
1 1 @F @F @F @F

@Var @RT(10)cMoveClose @RT(0) @T @F @DT @RT(4)DINT @RT(0) @T @T @BASIC 0 @F
@F @F
@T
@BEG_Attrib
0 @RT(2)51 @RT(44)close movement (for example shut off nozzle)
@END_Attrib
1 1 @F @F @F @F

@Var @RT(9)cMoveOpen @RT(0) @T @F @DT @RT(4)DINT @RT(0) @T @T @BASIC 0 @F
@F @F
@T
@BEG_Attrib
0 @RT(2)50 @RT(43)open movement (for example shut off nozzle)
@END_Attrib
1 1 @F @F @F @F

@END_Const

@BEG_Export

@BEG_Kind
@ALGORITHM_BLOCK @RT(15)ABMoveAutoPurge @STRUCTURED_TEXT
@RT(0) @RT(0) @RT(0)
@END_Kind

@BEG_Dcl
@RT(16)DclTreeContainer
7
@Var @RT(16)sv_MoveAutoPurge @RT(0) @T @T @DERIVED 0 @T @T @DT @RT(10)tsMoveData @RT(0) @T @T @UNKNOWN 0 @F
@F @F
@T
@BEG_Attrib
3 @RT(0) @RT(0) @RT(0)
@END_Attrib
1 8 @F @F @F @F

@Var @RT(16)sv_PurgeSettings @RT(0) @T @T @DERIVED 0 @T @T @DT @RT(15)tsPurgeSettings @RT(0) @T @T @UNKNOWN 0 @F
@F @F
@T
@BEG_Attrib
3 @RT(0) @RT(0) @RT(0)
@END_Attrib
1 8 @F @F @F @F

@Var @RT(17)sv_rScrewPosition @RT(0) @T @F @DT @RT(4)REAL @RT(0) @T @T @BASIC 0 @F
@F @F
@T
@BEG_Attrib
3 @RT(0) @RT(21)actual screw position @RT(0)
@END_Attrib
1 8 @F @F @F @F

@Var @RT(16)sv_ActPurgeTimes @RT(0) @T @T @DERIVED 0 @T @T @DT @RT(15)tsActPurgeTimes @RT(0) @T @T @UNKNOWN 0 @F
@F @F
@T
@BEG_Attrib
3 @RT(0) @RT(0) @RT(0)
@END_Attrib
1 8 @F @F @F @F

@Var @RT(18)sv_NumberOfDevices @RT(0) @T @T @DERIVED 0 @T @T @DT @RT(17)tyNumberOfDevices @RT(0) @T @T @UNKNOWN 0 @F
@F @F
@T
@BEG_Attrib
3 @RT(0) @RT(0) @RT(0)
@END_Attrib
1 8 @F @F @F @F

@Var @RT(11)sv_DeviceId @RT(0) @T @T @DERIVED 0 @T @T @DT @RT(10)tsDeviceId @RT(0) @T @T @UNKNOWN 0 @F
@F @F
@T
@BEG_Attrib
3 @RT(0) @RT(0) @RT(0)
@END_Attrib
1 8 @F @F @F @F

@Var @RT(14)evStartRequest @RT(0) @T @T @DERIVED 0 @T @T @DT @RT(15)tevStartRequest @RT(0) @T @T @UNKNOWN 0 @F
@F @F
@T
@BEG_Attrib
3 @RT(0) @RT(0) @RT(0)
@END_Attrib
1 7 @F @F @F @F

@END_Dcl

@END_Export

@BEG_Body

2

@BEG_Export

@BEG_Algo
@ALGORITHM @RT(9)aRegister @STRUCTURED_TEXT
@RT(0) @RT(0) @RT(0) @F @F
@END_Algo

@BEG_Dcl
@RT(16)DclTreeContainer
1
@Var @RT(18)abMovementRegister @RT(0) @T @T @DERIVED 0 @T @T @DT @RT(18)ABMovementRegister @RT(0) @T @T @UNKNOWN 0 @F
@F @F
@T
@BEG_Attrib
3 @RT(0) @RT(0) @RT(0)
@END_Attrib
1 0 @F @F @F @F

@END_Dcl

@END_Export

@BEG_Export

@BEG_Algo
@ALGORITHM @RT(4)aRun @SEQUENTIAL_FLOW_CHART
@RT(0) @RT(0) @RT(0) @F @F
@END_Algo

@BEG_Dcl
@RT(16)DclTreeContainer
16
@Var @RT(6)bReady @RT(0) @T @F @DT @RT(4)BOOL @RT(0) @T @T @BASIC 0 @F
@F @F
@T
@BEG_Attrib
3 @RT(0) @RT(0) @RT(0)
@END_Attrib
1 3 @F @F @F @F

@Var @RT(5)bStop @RT(0) @T @F @DT @RT(4)BOOL @RT(0) @T @T @BASIC 0 @F
@F @F
@T
@BEG_Attrib
3 @RT(0) @RT(0) @RT(0)
@END_Attrib
1 1 @F @F @F @F

@Var @RT(18)evStartRequestData @RT(0) @T @T @DERIVED 0 @T @T @DT @RT(19)tevStartRequestData @RT(0) @T @T @UNKNOWN 0 @F
@F @F
@T
@BEG_Attrib
3 @RT(0) @RT(0) @RT(0)
@END_Attrib
1 0 @F @F @F @F

@Var @RT(8)DeviceId @RT(0) @T @T @DERIVED 0 @T @T @DT @RT(10)tsDeviceId @RT(0) @T @T @UNKNOWN 0 @F
@F @F
@T
@BEG_Attrib
3 @RT(0) @RT(0) @RT(0)
@END_Attrib
1 0 @F @F @F @F

@Var @RT(12)fbCheckReady @RT(0) @T @T @DERIVED 0 @T @T @DT @RT(12)FBCheckReady @RT(0) @T @T @UNKNOWN 0 @F
@F @F
@T
@BEG_Attrib
3 @RT(0) @RT(0) @RT(0)
@END_Attrib
1 0 @F @F @F @F

@Var @RT(6)iCount @RT(0) @T @F @DT @RT(4)DINT @RT(0) @T @T @BASIC 0 @F
@F @F
@T
@BEG_Attrib
3 @RT(0) @RT(0) @RT(0)
@END_Attrib
1 0 @F @F @F @F

@Var @RT(6)fbStop @RT(0) @T @T @DERIVED 0 @T @T @DT @RT(6)FBStop @RT(0) @T @T @UNKNOWN 0 @F
@F @F
@T
@BEG_Attrib
3 @RT(0) @RT(0) @RT(0)
@END_Attrib
1 0 @F @F @F @F

@Var @RT(23)bShutOffNozzleAvailable @RT(0) @T @F @DT @RT(4)BOOL @RT(0) @T @T @BASIC 0 @F
@F @F
@T
@BEG_Attrib
3 @RT(0) @RT(0) @RT(0)
@END_Attrib
1 0 @F @F @F @F

@Var @RT(9)bInitDone @RT(0) @T @F @DT @RT(4)BOOL @RT(0) @T @T @BASIC 0 @F
@F @F
@T
@BEG_Attrib
3 @RT(0) @RT(0) @RT(0)
@END_Attrib
1 0 @F @F @F @F

@Var @RT(19)pbShutOffNozzleOpen @RT(0) @T @T @REFTO 0 @T @DT @RT(4)BOOL @RT(0) @T @T @BASIC 0 @F
@F @F
@T
@BEG_Attrib
3 @RT(0) @RT(0) @RT(0)
@END_Attrib
1 0 @F @F @F @F

@Var @RT(21)pbShutOffNozzleClosed @RT(0) @T @T @REFTO 0 @T @DT @RT(4)BOOL @RT(0) @T @T @BASIC 0 @F
@F @F
@T
@BEG_Attrib
3 @RT(0) @RT(0) @RT(0)
@END_Attrib
1 0 @F @F @F @F

@Var @RT(21)DeviceIdShutOffNozzle @RT(0) @T @T @DERIVED 0 @T @T @DT @RT(10)tsDeviceId @RT(0) @T @T @UNKNOWN 0 @F
@F @F
@T
@BEG_Attrib
3 @RT(0) @RT(0) @RT(0)
@END_Attrib
1 0 @F @F @F @F

@Var @RT(17)fbCheckPosReached @RT(0) @T @T @DERIVED 0 @T @T @DT @RT(17)FBCheckPosReached @RT(0) @T @T @UNKNOWN 0 @F
@F @F
@T
@BEG_Attrib
3 @RT(0) @RT(0) @RT(0)
@END_Attrib
1 0 @F @F @F @F

@Var @RT(13)fbDebugTrace2 @RT(0) @T @T @DERIVED 0 @T @T @DT @RT(13)FBDebugTrace2 @RT(0) @T @T @UNKNOWN 0 @F
@F @F
@T
@BEG_Attrib
3 @RT(0) @RT(0) @RT(0)
@END_Attrib
1 0 @F @F @F @F

@Var @RT(18)dTmpPurgePlastTime @RT(0) @T @T @RENAMED 0 @T @T @DT @RT(4)TIME @RT(0) @T @T @BASIC 0 @F
@F @F
@T
@BEG_Attrib
3 @RT(0) @RT(0) @RT(0)
@END_Attrib
1 0 @F @F @F @F

@Var @RT(18)rTmpPurgeDecompPos @RT(0) @T @F @DT @RT(4)REAL @RT(0) @T @T @BASIC 0 @F
@F @F
@T
@BEG_Attrib
3 @RT(0) @RT(0) @RT(0)
@END_Attrib
1 0 @F @F @F @F

@END_Dcl

@END_Export

@BEG_Body
@TL(15)
(**************************************** WARNING ********************************************
 *** The KEBA Kemro K2 System including software is not intended for safety control tasks! ***
 ***                       For further information see Comment tab!                        ***
 *********************************************************************************************)

// movement registration
sv_MoveAutoPurge.LockGroups[1] := cLockGroupHeatingNozzle;
sv_MoveAutoPurge.LockGroups[2] := cLockGroupSafetyGateNozzle;
sv_MoveAutoPurge.LockGroups[3] := cLockGroupSafetyGateMold;
sv_MoveAutoPurge.LockGroups[4] := cLockGroupMotor;

abMovementRegister.aRegister(@sv_MoveAutoPurge);

@END_Body

@@@BEG_Comment@@@
@TL(0)

@@@END_Comment@@@

@BEG_SfcBody
26 21 27

@BEG_SfcData 2
@StepSeq @RT(4)sseq @F 1
@Loop @RT(4)loop @F 2
@StepSeq @RT(4)sseq @F 11
@Step @RT(7)S_Start @F @T @F @F @RT(0) @F
@AcbCont @RT(7)unnamed @F 2
@Acb @RT(18)AInitShutOffNozzle @F @F @RT(1)P @RT(0) @F @F @F @F
@Acb @RT(6)AStart @F @T @RT(1)P @RT(0) @F @F @T @TL(4)
bReady := FALSE;
fbDebugTrace2(nDeviceState, 'AutoPurge started');
iCount := 0;

@F

@Trans @RT(6)TStart @F @T @F @F @T @F @TL(2)
TRUE

@RT(7)Trans21 @F
@Step @RT(6)Step17 @F @F @F @F @RT(0) @F
@AcbCont @RT(7)unnamed @F 0

@AltBranch @RT(3)alt @F 2
@TransSeq @RT(4)tseq @F 3
@Trans @RT(14)TShutOffNozzle @F @T @F @F @T @F @TL(2)
bShutOffNozzleAvailable

@RT(14)TShutOffNozzle @F
@Step @RT(19)S_OpenShutOffNozzle @F @F @F @F @RT(0) @F
@AcbCont @RT(7)unnamed @F 2
@Acb @RT(10)AStartOpen @F @F @RT(1)P @RT(0) @F @F @F @F
@Acb @RT(19)ACheckShutOffNozzle @F @T @RT(1)N @RT(0) @F @F @T @TL(2)
fbCheckReady(DeviceId := DeviceId);

@F

@AltBranch @RT(3)alt @F 2
@TransSeq @RT(4)tseq @F 1
@Trans @RT(18)TShutOffNozzleOpen @F @T @F @F @T @T @TL(2)
fbCheckReady.bReady AND pbShutOffNozzleOpen^

@RT(18)TShutOffNozzleOpen @F

@TransSeq @RT(4)tseq @F 2
@Trans @RT(6)TStop4 @F @T @F @F @T @T @TL(2)
bStop

@RT(6)TStop4 @F
@Goto @RT(6)S_Stop @F @F

@TransSeq @RT(4)tseq @F 1
@Trans @RT(16)TNoShutOffNozzle @F @T @T @F @T @F @TL(2)
NOT bShutOffNozzleAvailable

@RT(16)TNoShutOffNozzle @F

@Loop @RT(4)loop @F 2
@StepSeq @RT(4)sseq @F 7
@Step @RT(8)S_Inject @F @F @F @F @RT(0) @F
@AcbCont @RT(7)unnamed @F 2
@Acb @RT(12)AStartInject @F @T @RT(1)P @RT(0) @F @F @T @TL(9)
// send start request
DeviceId.CompId := cCompInjection;
DeviceId.IndexId := sv_DeviceId.IndexId;

evStartRequestData.DeviceId := DeviceId;
evStartRequestData.MoveDir := cMoveFwd;
evStartRequestData.MoveId := cMoveInjectPurge;
SET_EVENT(evStartRequest, evStartRequestData);

@F
@Acb @RT(17)ACheckInjectReady @F @T @RT(1)N @RT(0) @F @F @T @TL(2)
fbCheckReady(DeviceId := DeviceId);

@F

@AltBranch @RT(3)alt @F 2
@TransSeq @RT(4)tseq @F 1
@Trans @RT(12)TInjectReady @F @T @F @F @T @T @TL(3)
fbCheckReady.bReady AND
sv_rScrewPosition <= sv_PurgeSettings.InjectParams.rEndPos

@RT(12)TInjectReady @F

@TransSeq @RT(4)tseq @F 2
@Trans @RT(6)TStop1 @F @T @F @F @T @T @TL(2)
bStop

@RT(6)TStop1 @F
@Goto @RT(6)S_Stop @F @F

@Step @RT(8)S_Decomp @F @F @F @F @RT(0) @F
@AcbCont @RT(7)unnamed @F 2
@Acb @RT(12)AStartDecomp @F @T @RT(1)P @RT(0) @F @F @T @TL(13)
//copy decomp position to avoid wrongly detecting a error
//when the value changes while the movement is active
rTmpPurgeDecompPos := sv_PurgeSettings.DecompParams.rEndPos;

// send start request
DeviceId.CompId := cCompInjection;
DeviceId.IndexId := sv_DeviceId.IndexId;

evStartRequestData.DeviceId := DeviceId;
evStartRequestData.MoveDir := cMoveBwd;
evStartRequestData.MoveId := cMoveDecompPurge;
SET_EVENT(evStartRequest, evStartRequestData);

@F
@Acb @RT(17)ACheckDecompReady @F @T @RT(1)N @RT(0) @F @F @T @TL(2)
fbCheckReady(DeviceId := DeviceId);

@F

@AltBranch @RT(3)alt @F 2
@TransSeq @RT(4)tseq @F 1
@Trans @RT(12)TDecompReady @F @T @F @F @T @T @TL(3)
fbCheckReady.bReady AND
sv_rScrewPosition >= rTmpPurgeDecompPos

@RT(12)TDecompReady @F

@TransSeq @RT(4)tseq @F 2
@Trans @RT(6)TStop2 @F @T @F @F @T @T @TL(2)
bStop

@RT(6)TStop2 @F
@Goto @RT(6)S_Stop @F @F

@Step @RT(7)S_Plast @F @F @F @F @RT(0) @F
@AcbCont @RT(7)unnamed @F 2
@Acb @RT(11)AStartPlast @F @T @RT(1)P @RT(0) @F @F @T @TL(13)
//copy purge set time to avoid wrongly detecting a error
//when the value changes while the movement is active
dTmpPurgePlastTime := sv_PurgeSettings.PlastParams.dSetPlastTime;

// send start request
DeviceId.CompId := cCompInjection;
DeviceId.IndexId := sv_DeviceId.IndexId;

evStartRequestData.DeviceId := DeviceId;
evStartRequestData.MoveDir := cMoveBwd;
evStartRequestData.MoveId := cMovePlastPurge;
SET_EVENT(evStartRequest, evStartRequestData);

@F
@Acb @RT(16)ACheckPlastReady @F @T @RT(1)N @RT(0) @F @F @T @TL(2)
fbCheckReady(DeviceId := DeviceId);

@F

@AltBranch @RT(3)alt @F 2
@TransSeq @RT(4)tseq @F 1
@Trans @RT(11)TPlastReady @F @T @F @F @T @T @TL(3)
fbCheckReady.bReady AND
sv_ActPurgeTimes.dActPlastTime >= dTmpPurgePlastTime

@RT(11)TPlastReady @F

@TransSeq @RT(4)tseq @F 2
@Trans @RT(6)TStop3 @F @T @F @F @T @T @TL(2)
bStop

@RT(6)TStop3 @F
@Goto @RT(6)S_Stop @F @F

@Step @RT(14)S_CheckCounter @F @F @F @F @RT(0) @F
@AcbCont @RT(7)unnamed @F 1
@Acb @RT(8)ACounter @F @T @RT(1)P @RT(0) @F @F @T @TL(2)
iCount := iCount + 1;

@F

@Trans @RT(7)TRepeat @F @T @T @T @T @F @TL(2)
iCount < sv_PurgeSettings.iCount

@RT(7)TRepeat @F

@Trans @RT(6)TReady @F @T @F @F @T @F @TL(2)
iCount = sv_PurgeSettings.iCount

@RT(6)TReady @F
@Step @RT(11)S_CheckStop @F @F @F @F @RT(0) @F
@AcbCont @RT(7)unnamed @F 0

@AltBranch @RT(3)alt @F 2
@TransSeq @RT(4)tseq @F 3
@Trans @RT(5)TStop @F @T @F @F @T @F @TL(2)
bStop

@RT(5)TStop @F
@Step @RT(6)S_Stop @F @F @T @F @RT(0) @F
@AcbCont @RT(7)unnamed @F 2
@Acb @RT(19)AStopActiveMovement @F @T @RT(1)P @RT(0) @F @F @T @TL(3)
//stop actual active movement
fbStop(DeviceId := DeviceId);

@F
@Acb @RT(17)AStoppedMoveReady @F @T @RT(1)N @RT(0) @F @F @T @TL(2)
fbCheckReady(DeviceId := DeviceId);

@F

@Trans @RT(19)TStoppedDeviceReady @F @T @F @F @T @T @TL(2)
fbCheckReady.bReady

@RT(19)TStoppedDeviceReady @F

@TransSeq @RT(4)tseq @F 1
@Trans @RT(7)TNoStop @F @T @T @F @T @F @TL(2)
NOT bStop

@RT(7)TNoStop @F

@Step @RT(6)Step27 @F @F @F @F @RT(0) @F
@AcbCont @RT(7)unnamed @F 0

@AltBranch @RT(3)alt @F 2
@TransSeq @RT(4)tseq @F 3
@Trans @RT(7)Trans36 @F @T @F @F @T @F @TL(2)
bShutOffNozzleAvailable

@RT(7)Trans36 @F
@Step @RT(20)S_CloseShutOffNozzle @F @F @F @F @RT(0) @F
@AcbCont @RT(7)unnamed @F 2
@Acb @RT(11)AStartClose @F @F @RT(1)P @RT(0) @F @F @F @F
@Acb @RT(13)ACheckShutOff @F @T @RT(1)N @RT(0) @F @F @T @TL(2)
fbCheckReady(DeviceId := DeviceId);

@F

@Trans @RT(19)TShutOffNozzleReady @F @T @F @F @T @T @TL(2)
fbCheckReady.bReady

@RT(20)TShutOffNozzleClosed @F

@TransSeq @RT(4)tseq @F 1
@Trans @RT(7)Trans37 @F @T @T @F @T @F @TL(2)
NOT bShutOffNozzleAvailable

@RT(7)Trans37 @F

@Step @RT(7)S_Ready @F @F @F @F @RT(0) @F
@AcbCont @RT(7)unnamed @F 1
@Acb @RT(6)AReady @F @T @RT(1)P @RT(0) @F @F @T @TL(3)
bReady := TRUE;
fbDebugTrace2(nDeviceState, 'AutoPurge ready');

@F

@Trans @RT(7)Trans12 @F @T @T @T @T @T @TL(2)
TRUE

@RT(7)Trans12 @F

@END_SfcData
@SaActions 3
@SaText @RT(18)AInitShutOffNozzle 1 @TL(24)
//check if shut off nozzle is available
IF NOT bInitDone THEN
   bShutOffNozzleAvailable := sv_NumberOfDevices[cCompShutOffNozzle] = sv_DeviceId.IndexId;
END_IF;

IF bShutOffNozzleAvailable AND NOT bInitDone THEN
   //get pos reached flags of shut off nozzle
   DeviceIdShutOffNozzle.CompId := cCompShutOffNozzle;
   DeviceIdShutOffNozzle.IndexId := sv_DeviceId.IndexId;

   fbCheckPosReached.DeviceId := DeviceIdShutOffNozzle;
   fbCheckPosReached.MoveDir := cMoveClose;
   fbCheckPosReached.MoveId := cMoveClose;
   fbCheckPosReached();
   pbShutOffNozzleClosed := fbCheckPosReached.pbPosReached;

   fbCheckPosReached.MoveDir := cMoveOpen;
   fbCheckPosReached.MoveId := cMoveOpen;
   fbCheckPosReached();
   pbShutOffNozzleOpen := fbCheckPosReached.pbPosReached;
END_IF;

bInitDone := TRUE;

@SaText @RT(10)AStartOpen 1 @TL(13)
(**************************************** WARNING ********************************************
 *** The KEBA Kemro K2 System including software is not intended for safety control tasks! ***
 ***                       For further information see Comment tab!                        ***
 *********************************************************************************************)

// send start request
DeviceId := DeviceIdShutOffNozzle;

evStartRequestData.DeviceId := DeviceId;
evStartRequestData.MoveDir := cMoveOpen;
evStartRequestData.MoveId := cMoveOpen;
SET_EVENT(evStartRequest, evStartRequestData);

@SaText @RT(11)AStartClose 1 @TL(12)
(**************************************** WARNING ********************************************
 *** The KEBA Kemro K2 System including software is not intended for safety control tasks! ***
 ***                       For further information see Comment tab!                        ***
 *********************************************************************************************)

// send start request
DeviceId := DeviceIdShutOffNozzle;
evStartRequestData.DeviceId := DeviceId;
evStartRequestData.MoveDir := cMoveClose;
evStartRequestData.MoveId := cMoveClose;
SET_EVENT(evStartRequest, evStartRequestData);

@SaTrans 0
@SaExits 0
@END_SfcBody

@@@BEG_Comment@@@
@TL(0)

@@@END_Comment@@@
@END_Body

@END_Contents

(* ---- ABMovementAdmin.pu ---- *)
IMPORT_OVER_LISTFILE
 tsMoveCtrl
, ABMoveAutoPurge
, tsPurgeSettings
, tsActPurgeTimes
, TON
, R_TRIG

END_IMPORT

ALGORITHM_BLOCK ABMovementAdmin #DUMMY_EDIT_BLOCK

SYSTEM_VAR
 sv_bInitStart : BOOL;
 sv_bDeviceStart : BOOL (* Start Device *);
 sv_PurgeSettings : tsPurgeSettings;
 sv_ActPurgeTimes : tsActPurgeTimes (* actual times of purge movement *);
 sv_bFALSE : BOOL;
END_VAR

SYSTEM_OBJECT
 PU_Task_7 : TASK;
 TaskMid : TASK;
 erAutoPurgeTimeout : ALARM;
END_OBJECT

VAR_EXTERNAL
 g_MoveCtrl : tsMoveCtrl;
END_VAR

VAR
 abMoveAutoPurge : ABMoveAutoPurge;
END_VAR

(*
Calls the registration-algo of every movementblock after the deviceregistration succeeded(sv_bInitStart->true)

*)

POSTUPDATE_ALGORITHM pInitStart ON PU_Task_7 WITH sv_bInitStart

#BEGIN_EDIT_BLOCK
(**************************************** WARNING ********************************************
 *** The KEBA Kemro K2 System including software is not intended for safety control tasks! ***
 ***                       For further information see Comment tab!                        ***
 *********************************************************************************************)

IF sv_bInitStart THEN
    //Register Movement
    abMoveAutoPurge.aRegister();
END_IF;

;#END_EDIT_BLOCK END_ALGORITHM

(*
Starts the algo paRun when sv_bDeviceStart is set by ABControl.
*)

POSTUPDATE_ALGORITHM pDeviceStart ON PU_Task_7 WITH sv_bDeviceStart

#BEGIN_EDIT_BLOCK
(**************************************** WARNING ********************************************
 *** The KEBA Kemro K2 System including software is not intended for safety control tasks! ***
 ***                       For further information see Comment tab!                        ***
 *********************************************************************************************)

IF sv_bDeviceStart THEN
   //start device
   START_PROCESS_ALGORITHM(paRun);
END_IF;

;#END_EDIT_BLOCK END_ALGORITHM

(*
Calls depending on the MoveId and MoveDir the movementblock. g_MoveCtrl.MoveId/MoveDir are set by the Block ABControl after
evStart was received. The movement-block has to be called until the it returns abMoveXxx.aRun.bReady.
In case of hydraulic movements the output-request has to be done before starting the movement.
*)

PROCESS_ALGORITHM paRun ON TaskMid

VAR_TEMP
 b : BOOL;
END_VAR

VAR
 fbPurgeTimer : TON;
 bTimeOut : BOOL;
 fbRTrigTimeOut : R_TRIG;
END_VAR

(* IecGraph-Code *)

(* init step *)
INITIAL_STEP S_Start:
AResetTimeout (P);
END_STEP

ACTION AResetTimeout: #BEGIN_EDIT_BLOCK
b := WRITE_SV_DIRECT(sv_bDeviceStart, sv_bFALSE);
bTimeOut := FALSE;

;#END_EDIT_BLOCK END_ACTION (*AResetTimeout*)

(* steps *)
STEP S_Purge:
AResetTimer (P);
AAutoPurge (N);
ACheckTimeout (N);
END_STEP

ACTION AResetTimer: #BEGIN_EDIT_BLOCK
fbPurgeTimer(IN := FALSE,
             PT := sv_PurgeSettings.dMaxPurgeTime);

;#END_EDIT_BLOCK END_ACTION (*AResetTimer*)
ACTION ACheckTimeout: #BEGIN_EDIT_BLOCK
fbPurgeTimer(IN := TRUE,
             PT := sv_PurgeSettings.dMaxPurgeTime);

sv_ActPurgeTimes.dActPurgeTime := fbPurgeTimer.ET;
bTimeOut := fbPurgeTimer.Q;

fbRTrigTimeOut(CLK := bTimeOut);
IF fbRTrigTimeOut.Q THEN
    SET_ALARM(Name := erAutoPurgeTimeout);
END_IF;

;#END_EDIT_BLOCK END_ACTION (*ACheckTimeout*)
STEP READY:
AReady (P);
END_STEP

ACTION AReady: #BEGIN_EDIT_BLOCK
g_MoveCtrl.bReady := TRUE;
IF NOT sv_bDeviceStart THEN
   STOP_PROCESS_ALGORITHM();
END_IF;
;#END_EDIT_BLOCK END_ACTION (*AReady*)

(* transitions *)
GO_ON_TRANSITION TStart (* Trans9 *) FROM S_Start TO S_Purge :=  #BEGIN_EDIT_BLOCK
TRUE
;#END_EDIT_BLOCK
END_TRANSITION

TRANSITION TPurgeReady (* Trans1 *) FROM S_Purge TO READY :=  #BEGIN_EDIT_BLOCK
abMoveAutoPurge.aRun.bReady;
;#END_EDIT_BLOCK
END_TRANSITION

TRANSITION Trans8 (* Trans8 *) FROM READY TO S_Start :=  #BEGIN_EDIT_BLOCK
TRUE
;#END_EDIT_BLOCK
END_TRANSITION

(* end IecGraph-Code *)
(* sfc-code *)

(* stand alone actions *)
ACTION AAutoPurge: #BEGIN_EDIT_BLOCK
(**************************************** WARNING ********************************************
 *** The KEBA Kemro K2 System including software is not intended for safety control tasks! ***
 ***                       For further information see Comment tab!                        ***
 *********************************************************************************************)

abMoveAutoPurge.aRun(bStop := g_MoveCtrl.bStop OR bTimeOut);

;#END_EDIT_BLOCK END_ACTION (*AAutoPurge*)
(* end sfc-code *)

END_ALGORITHM

END_ALGORITHM_BLOCK

#END_OF_IEC_PART

@Puma @IecEditor 6 68 @Pou 25
@@@BEG_Comment@@@

@@@END_Comment@@@

@BEG_Contents

@BEG_Func
@RT(17)FuncTreeContainer
0
@END_Func

@BEG_Const
@RT(18)ConstTreeContainer
0
@END_Const

@BEG_Export

@BEG_Kind
@ALGORITHM_BLOCK @RT(15)ABMovementAdmin @STRUCTURED_TEXT
@RT(0) @RT(0) @RT(0)
@END_Kind

@BEG_Dcl
@RT(16)DclTreeContainer
10
@Var @RT(13)sv_bInitStart @RT(0) @T @F @DT @RT(4)BOOL @RT(0) @T @T @BASIC 0 @F
@F @F
@T
@BEG_Attrib
3 @RT(0) @RT(0) @RT(0)
@END_Attrib
1 8 @F @F @F @F

@Var @RT(15)sv_bDeviceStart @RT(0) @T @F @DT @RT(4)BOOL @RT(0) @T @T @BASIC 0 @F
@F @F
@T
@BEG_Attrib
3 @RT(0) @RT(12)Start Device @RT(0)
@END_Attrib
1 8 @F @F @F @F

@Var @RT(10)g_MoveCtrl @RT(0) @T @T @DERIVED 0 @T @T @DT @RT(10)tsMoveCtrl @RT(0) @T @T @UNKNOWN 0 @F
@F @F
@T
@BEG_Attrib
3 @RT(0) @RT(0) @RT(0)
@END_Attrib
1 6 @F @F @F @F

@Var @RT(9)PU_Task_7 @RT(0) @T @T @RENAMED 0 @T @T @DT @RT(4)TASK @RT(0) @T @T @BASIC 0 @F
@F @F
@T
@BEG_Attrib
3 @RT(0) @RT(0) @RT(0)
@END_Attrib
1 7 @F @F @F @F

@Var @RT(15)abMoveAutoPurge @RT(0) @T @T @DERIVED 0 @T @T @DT @RT(15)ABMoveAutoPurge @RT(0) @T @T @UNKNOWN 0 @F
@F @F
@T
@BEG_Attrib
3 @RT(0) @RT(0) @RT(0)
@END_Attrib
1 0 @F @F @F @F

@Var @RT(16)sv_PurgeSettings @RT(0) @T @T @DERIVED 0 @T @T @DT @RT(15)tsPurgeSettings @RT(0) @T @T @UNKNOWN 0 @F
@F @F
@T
@BEG_Attrib
3 @RT(0) @RT(0) @RT(0)
@END_Attrib
1 8 @F @F @F @F

@Var @RT(7)TaskMid @RT(0) @T @T @RENAMED 0 @T @T @DT @RT(4)TASK @RT(0) @T @T @BASIC 0 @F
@F @F
@T
@BEG_Attrib
3 @RT(0) @RT(0) @RT(0)
@END_Attrib
1 7 @F @F @F @F

@Var @RT(18)erAutoPurgeTimeout @RT(0) @T @F @DT @RT(5)ALARM @RT(0) @T @T @BASIC 0 @F
@F @F
@T
@BEG_Attrib
3 @RT(0) @RT(0) @RT(0)
@END_Attrib
1 7 @F @F @F @F

@Var @RT(16)sv_ActPurgeTimes @RT(0) @T @T @DERIVED 0 @T @T @DT @RT(15)tsActPurgeTimes @RT(0) @T @T @UNKNOWN 0 @F
@F @F
@T
@BEG_Attrib
3 @RT(0) @RT(30)actual times of purge movement @RT(0)
@END_Attrib
1 8 @F @F @F @F

@Var @RT(9)sv_bFALSE @RT(0) @T @F @DT @RT(4)BOOL @RT(0) @T @T @BASIC 0 @F
@F @F
@T
@BEG_Attrib
3 @RT(0) @RT(0) @RT(0)
@END_Attrib
1 8 @F @F @F @F

@END_Dcl

@END_Export

@BEG_Body

3

@BEG_Export

@BEG_Algo
@POSTUPDATE_ALGORITHM @RT(10)pInitStart @STRUCTURED_TEXT
@RT(0) @RT(13)sv_bInitStart @RT(9)PU_Task_7 @F @F
@END_Algo

@BEG_Dcl
@RT(16)DclTreeContainer
0
@END_Dcl

@END_Export

@BEG_Export

@BEG_Algo
@POSTUPDATE_ALGORITHM @RT(12)pDeviceStart @STRUCTURED_TEXT
@RT(0) @RT(15)sv_bDeviceStart @RT(9)PU_Task_7 @F @F
@END_Algo

@BEG_Dcl
@RT(16)DclTreeContainer
0
@END_Dcl

@END_Export

@BEG_Export

@BEG_Algo
@PROCESS_ALGORITHM @RT(5)paRun @SEQUENTIAL_FLOW_CHART
@RT(0) @RT(0) @RT(7)TaskMid @F @F
@END_Algo

@BEG_Dcl
@RT(16)DclTreeContainer
4
@Var @RT(12)fbPurgeTimer @RT(0) @T @T @DERIVED 0 @T @T @DT @RT(3)TON @RT(0) @T @T @UNKNOWN 0 @F
@F @F
@T
@BEG_Attrib
3 @RT(0) @RT(0) @RT(0)
@END_Attrib
1 0 @F @F @F @F

@Var @RT(8)bTimeOut @RT(0) @T @F @DT @RT(4)BOOL @RT(0) @T @T @BASIC 0 @F
@F @F
@T
@BEG_Attrib
3 @RT(0) @RT(0) @RT(0)
@END_Attrib
1 0 @F @F @F @F

@Var @RT(14)fbRTrigTimeOut @RT(0) @T @T @RENAMED 0 @T @T @DT @RT(6)R_TRIG @RT(0) @T @T @UNKNOWN 0 @F
@F @F
@T
@BEG_Attrib
3 @RT(0) @RT(0) @RT(0)
@END_Attrib
1 0 @F @F @F @F

@Var @RT(1)b @RT(0) @T @F @DT @RT(4)BOOL @RT(0) @T @T @BASIC 0 @F
@F @F
@T
@BEG_Attrib
3 @RT(0) @RT(0) @RT(0)
@END_Attrib
1 4 @F @F @F @F

@END_Dcl

@END_Export

@BEG_Body
@TL(10)
(**************************************** WARNING ********************************************
 *** The KEBA Kemro K2 System including software is not intended for safety control tasks! ***
 ***                       For further information see Comment tab!                        ***
 *********************************************************************************************)

IF sv_bInitStart THEN
    //Register Movement
    abMoveAutoPurge.aRegister();
END_IF;

@END_Body

@@@BEG_Comment@@@
@TL(2)
Calls the registration-algo of every movementblock after the deviceregistration succeeded(sv_bInitStart->true)

@@@END_Comment@@@

@BEG_Body
@TL(10)
(**************************************** WARNING ********************************************
 *** The KEBA Kemro K2 System including software is not intended for safety control tasks! ***
 ***                       For further information see Comment tab!                        ***
 *********************************************************************************************)

IF sv_bDeviceStart THEN
   //start device
   START_PROCESS_ALGORITHM(paRun);
END_IF;

@END_Body

@@@BEG_Comment@@@
@TL(1)
Starts the algo paRun when sv_bDeviceStart is set by ABControl.
@@@END_Comment@@@

@BEG_SfcBody
23 18 21

@BEG_SfcData 2
@StepSeq @RT(4)sseq @F 1
@Loop @RT(4)loop @F 2
@StepSeq @RT(3)seq @F 5
@Step @RT(7)S_Start @F @T @F @F @RT(0) @F
@AcbCont @RT(7)unnamed @F 1
@Acb @RT(13)AResetTimeout @F @T @RT(1)P @RT(0) @F @F @T @TL(3)
b := WRITE_SV_DIRECT(sv_bDeviceStart, sv_bFALSE);
bTimeOut := FALSE;

@F

@Trans @RT(6)TStart @F @T @F @F @T @F @TL(2)
TRUE

@RT(6)Trans9 @F
@Step @RT(7)S_Purge @F @F @F @F @RT(0) @F
@AcbCont @RT(7)unnamed @F 3
@Acb @RT(11)AResetTimer @F @T @RT(1)P @RT(0) @F @F @T @TL(3)
fbPurgeTimer(IN := FALSE,
             PT := sv_PurgeSettings.dMaxPurgeTime);

@F
@Acb @RT(10)AAutoPurge @F @F @RT(1)N @RT(0) @F @F @F @F
@Acb @RT(13)ACheckTimeout @F @T @RT(1)N @RT(0) @F @F @T @TL(13)
fbPurgeTimer(IN := TRUE,
             PT := sv_PurgeSettings.dMaxPurgeTime);

sv_ActPurgeTimes.dActPurgeTime := fbPurgeTimer.ET;
bTimeOut := fbPurgeTimer.Q;

fbRTrigTimeOut(CLK := bTimeOut);
IF fbRTrigTimeOut.Q THEN
    SET_ALARM(Name := erAutoPurgeTimeout);
END_IF;

@F

@Trans @RT(11)TPurgeReady @F @T @F @F @T @T @TL(2)
abMoveAutoPurge.aRun.bReady;

@RT(6)Trans1 @F
@Step @RT(5)READY @F @F @F @F @RT(0) @F
@AcbCont @RT(7)unnamed @F 1
@Acb @RT(6)AReady @F @T @RT(1)P @RT(0) @F @F @T @TL(4)
g_MoveCtrl.bReady := TRUE;
IF NOT sv_bDeviceStart THEN
   STOP_PROCESS_ALGORITHM();
END_IF;
@F

@Trans @RT(6)Trans8 @F @T @T @T @T @T @TL(2)
TRUE

@RT(6)Trans8 @F

@END_SfcData
@SaActions 1
@SaText @RT(10)AAutoPurge 1 @TL(7)
(**************************************** WARNING ********************************************
 *** The KEBA Kemro K2 System including software is not intended for safety control tasks! ***
 ***                       For further information see Comment tab!                        ***
 *********************************************************************************************)

abMoveAutoPurge.aRun(bStop := g_MoveCtrl.bStop OR bTimeOut);

@SaTrans 0
@SaExits 0
@END_SfcBody

@@@BEG_Comment@@@
@TL(3)
Calls depending on the MoveId and MoveDir the movementblock. g_MoveCtrl.MoveId/MoveDir are set by the Block ABControl after
evStart was received. The movement-block has to be called until the it returns abMoveXxx.aRun.bReady.
In case of hydraulic movements the output-request has to be done before starting the movement.
@@@END_Comment@@@
@END_Body

@END_Contents
